SUBAPPLICATION Uebung_004a6_AX (* Toggle Flip-Flop mit IE und E_REND (Rendezvous) *)
  (* Standard: 61499-2; Description: Copyright (c) 2023 Meisterschulen am Ostbahnhof This program and the accompanying materials are made available under the terms of the Eclipse Public License 2.0 which is available at https://www.eclipse.org/legal/epl-2.0/ SPDX-License-Identifier: EPL-2.0 *)
  (* Version 1.0, 2023-10-23, Franz Höpfinger, Meisterschulen am Ostbahnhof *)
  PACKAGE Uebungen;
  IMPORT logiBUS::io::DI::logiBUS_DI::Input_I1;
  IMPORT logiBUS::io::DI::logiBUS_DI::Input_I2;
  IMPORT logiBUS::io::DI::logiBUS_DI::Input_I3;
  IMPORT logiBUS::io::DI::logiBUS_DI_Events::BUTTON_SINGLE_CLICK;
  IMPORT logiBUS::io::DQ::logiBUS_DO::Output_Q1;
  IMPORT logiBUS::io::DQ::logiBUS_DO::Output_Q2;
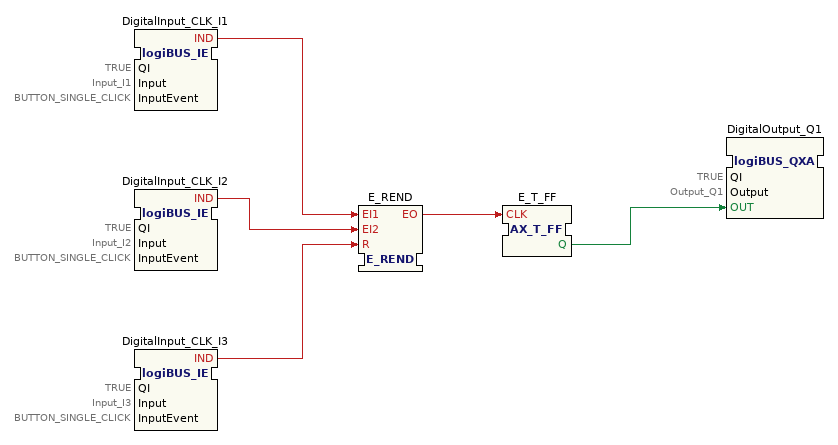
  FBS
    DigitalOutput_Q1 : logiBUS::io::DQ::logiBUS_QXA(QI := TRUE, Output := Output_Q1);
    DigitalInput_CLK_I1 : logiBUS::io::DI::logiBUS_IE(QI := TRUE, Input := Input_I1, InputEvent := BUTTON_SINGLE_CLICK);
    E_T_FF : adapter::events::unidirectional::AX_T_FF;
    E_REND : iec61499::events::E_REND;
    DigitalInput_CLK_I2 : logiBUS::io::DI::logiBUS_IE(QI := TRUE, Input := Input_I2, InputEvent := BUTTON_SINGLE_CLICK);
    DigitalInput_CLK_I3 : logiBUS::io::DI::logiBUS_IE(QI := TRUE, Input := Input_I3, InputEvent := BUTTON_SINGLE_CLICK);
  END_FBS
  EVENT_CONNECTIONS
    DigitalInput_CLK_I1.IND TO E_REND.EI1;
    DigitalInput_CLK_I2.IND TO E_REND.EI2;
    DigitalInput_CLK_I3.IND TO E_REND.R;
    E_REND.EO TO E_T_FF.CLK;
  END_CONNECTIONS
  ADAPTER_CONNECTIONS
    E_T_FF.Q TO DigitalOutput_Q1.OUT;
  END_CONNECTIONS
END_SUBAPPLICATION
